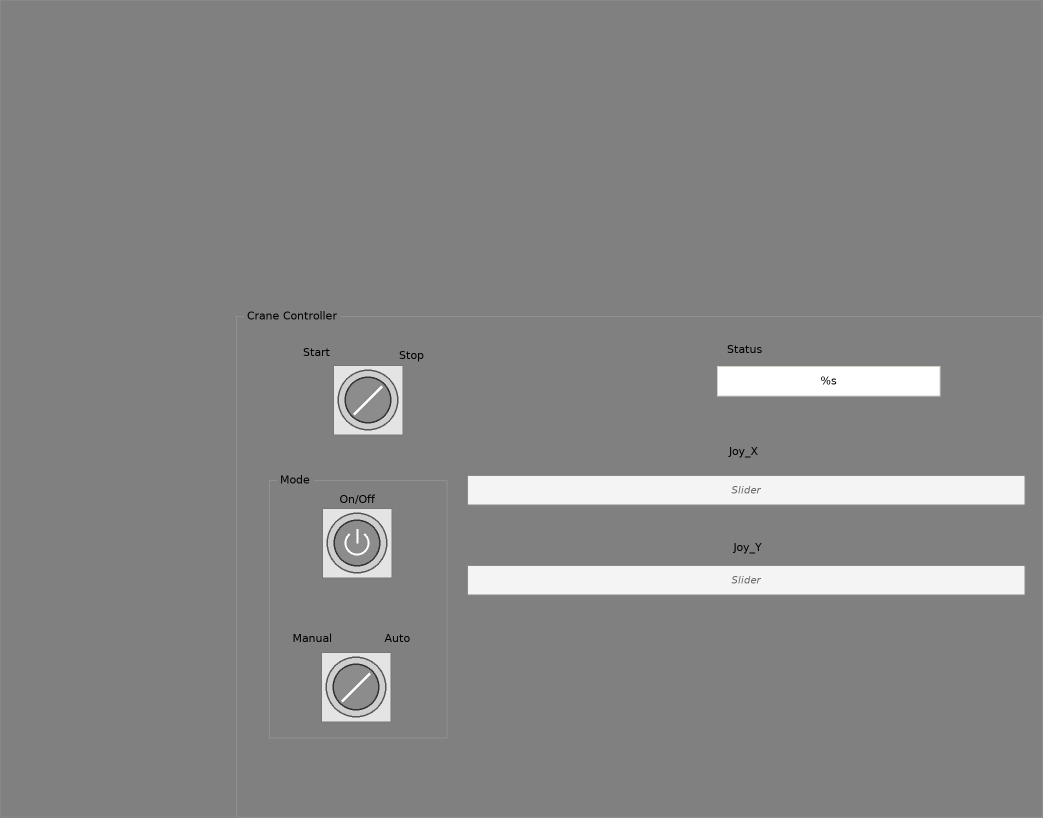
VISUALIZATION CraneController  // 1043x818
    GroupBox (236,308 807x510), "Crane Controller"
        GroupBox (33,164 178x266), "Mode"
            Label (61,14 55x27), "On/Off"
            Label (101,153 55x27), "Auto"
            PowerSwitch (53,36 70x70), variable: G_HMI.stHMIVaribles.bOn, behaviour: TOGGLE, style: Switch-PowerSwitch-Gray
            RotarySwitch (52,180 70x70), variable: G_HMI.stHMIVaribles.bAuto, behaviour: TOGGLE, style: Switch-RotarySwitch-Gray
            Label (16,153 55x27), "Manual"
        Textfield (481,58 223x30), "%s", text variable: G_HMI.stHMIVaribles.sStatus
        Label (484,226 55x27), "Joy_Y"
        Label (480,130 55x27), "Joy_X"
        Slider (231,257 558x30), variable: G_HMI.stHMIVaribles.fJoyY, scale 0..100
        Label (481,28 55x27), "Status"
        RotarySwitch (97,57 70x70), variable: G_HMI.stHMIVaribles.bStart, behaviour: TOGGLE, style: Switch-RotarySwitch-Gray
        Label (53,31 55x27), "Start"
        Label (148,34 55x27), "Stop"
        Slider (231,167 558x30), variable: G_HMI.stHMIVaribles.fJoyX, scale 0..32767
END_VISUALIZATION

(* stored: Version 1.1.0.1, ProductVersion 3.1.4024.12
   Visu CraneController: Id {563b52cb-7a03-4657-9928-2af245d11a46} *)
